(* CODESYS project wago_750-673_stepper_simple_v0.0.1.ecp

Project tree, tasks and I/O mapping:
  PFC100_2ETH : 750-8101 PFC100 CS 2ETH, WAGO, order no. 0750-8101, version 5.11.1.16
    application Application
      libraries: ; WagoAppStepper, * (WAGO); VisuDialogs, * (System)
      task PLC_Task (cyclic, interval t#50ms, priority 15) calls PLC_PRG
      task VISU_TASK (cyclic, interval 100 ms, priority 15) calls VisuElems.Visu_Prg
      program PLC_PRG [ST]
      visualisation Visualization
    DeviceAdapter
    Kbus : Kbus, WAGO, version 1.4.0.2
        unmapped channels: K-BUS diagnostics
      Servo_Stepper_Controller_55_VDC_7_5A : 0750-0673, WAGO, order no. 0750-0673, version 0.0.0.19
          settings: K-BUS Module slot index = 1
          unmapped channels: status byte S0, speed, process value, status byte S3, status byte S2, status byte S1, control byte C0, speed, acceleration, process value, control byte C3, control byte C2, control byte C1
        DeviceAdapter
    MODBUS
      MODBUS : MODBUS, WAGO, order no. n/a, version 1.1.1.15
    Serial
  text list GlobalTextList
*)

// PFC100_2ETH/Application/PLC_PRG
PROGRAM PLC_PRG
VAR
	fb673				: WagoAppStepper.FbStepperControlBasic;
	fb673_Velocity		: WagoAppStepper.FbMoveVelocity_2;
	xStepperEnable		: BOOL;
	eStepperJobType		: eMode;
	xStepperDirPos		: BOOL;
	xStepperDirNeg		: BOOL;
	iStepperSpeed		: INT := 10000;
	wStepperAccel		: WORD := 15000;
	wStepperDecel		: WORD := 15000;
	diStepperPosition	: DINT;
	xStepperStart		: BOOL;
	xStepperErrorRst	: BOOL;
	xStepperStop		: BOOL;
	xStepperJobFinished	: BOOL;
	xStepperIsBusy		: BOOL;
	xStepperError		: BOOL;
	oStepperStatus		: WagoSysErrorBase.FbResult;
	eStepperErrorCodes	: eStatus;
	diStepperActualPosition: DINT;
	iStepperActualSpeed	: INT;
	xStepperMbxActive	: BOOL;
	xStepperResetWarning: BOOL;
	xStepperMoveVel		: BOOL;
	xStepperInVel		: BOOL;
	xStepperMoveVelBusy	: BOOL;
	xStepperVelError	: BOOL;
	oStepperVelStatus	: WagoSysErrorBase.FbResult;
	
	// mode selection
	xStepperMoveAbsolute	: BOOL := TRUE;
	xStepperMoveRelative	: BOOL;
	xStepperMoveHome		: BOOL;
	xStepperMoveJog			: BOOL;
	xStepperProg			: BOOL;
	xStepperMoveTorqueEdge	: BOOL;
	xStepperMoveTorqueLevel	: BOOL;
	xStepperSetPos			: BOOL;
END_VAR

eStepperJobType := WagoAppStepper.FuModeSelect(
	xMoveAbsoluteRequest:= xStepperMoveAbsolute, 
	xMoveRelativeRequest:= xStepperMoveRelative, 
	xHomingRequest:= xStepperMoveHome, 
	xJoggingRequest:= xStepperMoveJog, 
	xVelocityCtrlRequest:= xStepperMoveVel, 
	xDrivePrgRequest:= xStepperProg, 
	xTorqueEdge:= xStepperMoveTorqueEdge, 
	xTorqueLevel:= xStepperMoveTorqueLevel, 
	xSetPosition:= xStepperSetPos);

fb673(
	xEnable:= xStepperEnable, 
	I_Port:= IoConfig_Globals.Servo_Stepper_Controller_55_VDC_7_5A, 
	eJobType:= eStepperJobType, 
	xDirPos:= xStepperDirPos, 
	xDirNeg:= xStepperDirNeg, 
	iSpeed:= iStepperSpeed, 
	wAcceleration:= wStepperAccel, 
	wDeceleration:= wStepperDecel, 
	diPosition:= diStepperPosition, 
	xTriggerStart:= xStepperStart, 
	xTriggerErrorReset:= xStepperErrorRst, 
	xStop:= xStepperStop, 
	xJobFinished=> xStepperJobFinished, 
	xBusy=> xStepperIsBusy, 
	xError=> xStepperError, 
	oStatus=> oStepperStatus, 
	eErrorCodes=> eStepperErrorCodes, 
	diActualPosition=> diStepperActualPosition, 
	iActualSpeed=> iStepperActualSpeed, 
	xMailboxActive=> xStepperMbxActive, 
	xResetWarning=> xStepperResetWarning);

END_PROGRAM

// PFC100_2ETH/Application/Visualization
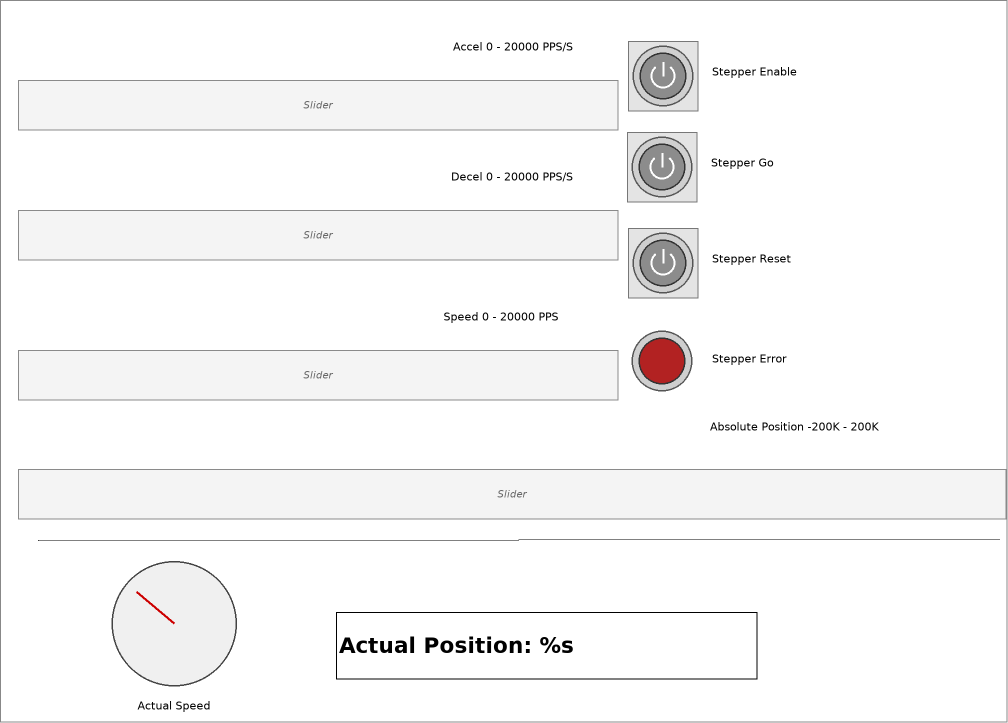
VISUALIZATION Visualization  // 1008x723
    Slider (18,80 600x50), variable: PLC_PRG.wStepperAccel, scale 0..20000
    Label (426,32 150x30), "Accel 0 - 20000 PPS/S"
    Slider (18,210 600x50), variable: PLC_PRG.wStepperDecel, scale 0..20000
    Label (426,162 150x30), "Decel 0 - 20000 PPS/S"
    Slider (18,350 600x50), variable: PLC_PRG.iStepperSpeed, scale 0..20000
    Label (426,302 150x30), "Speed 0 - 20000 PPS"
    PowerSwitch (628,41 70x70), variable: PLC_PRG.xStepperEnable, behaviour: TOGGLE, style: Switch-PowerSwitch-Gray
    Label (709,57 150x30), "Stepper Enable"
    PowerSwitch (627,132 70x70), variable: PLC_PRG.xStepperStart, behaviour: TOGGLE, style: Switch-PowerSwitch-Gray
    Label (708,148 150x30), "Stepper Go"
    PowerSwitch (628,228 70x70), variable: PLC_PRG.xStepperErrorRst, behaviour: TOGGLE, style: Switch-PowerSwitch-Gray
    Label (709,244 150x30), "Stepper Reset"
    Lamp1 (627,326 70x70), variable: PLC_PRG.xStepperError, style: Lamp-Lamp1-Red
    Label (709,344 150x30), "Stepper Error"
    Line (38,540) (999,539)
    Meter180 (49,561 250x125), value: PLC_PRG.iStepperActualSpeed, style: Meter-Meter180-Gray, scale format: %.0f, scale 0..20000
    Label (62,691 224x30), "Actual Speed"
    Rectangle (336,612 421x67), "Actual Position: %s", text variable: PLC_PRG.diStepperActualPosition
    Slider (18,469 988x50), variable: PLC_PRG.diStepperPosition, scale -200000..200000
    Label (673,412 243x30), "Absolute Position -200K - 200K"
END_VISUALIZATION
